FUNCTION_BLOCK FB_TON_1
VAR_INPUT
	IN 			: BOOL;
	PT			: TIME	:= T#0ms;
	ET 			: TIME	:= T#0ms;
END_VAR
VAR_OUTPUT
	Q			: BOOL;
END_VAR
VAR
END_VAR

IF IN THEN
	ET := ET + CYCLE_TIME_IN_MS;
	IF ET > PT THEN
		Q := TRUE;
	END_IF
ELSE
	ET := T#0ms;
	Q := FALSE;
END_IF

END_FUNCTION_BLOCK

(* stored: Version 1.1.0.1, ProductVersion 3.1.4022.12
   POU FB_TON_1: Id {41d316f8-2c52-4c58-bb5a-b4376f9ea1ca}, SpecialFunc None *)
